{attribute 'qualified_only'}
VAR_GLOBAL
	Sc1:BOOL;
	Sc2:BOOL;
	Busc1:BOOL;
	Busc2:BOOL;
	Backup_safety_trip:BOOL;
	Main_safety_trip:BOOL;
	Lily_func_trip:BOOL;
	Lily_app_fault:BOOL;
	Backup_control_trip:BOOL;
	Control_trip:BOOL;
	Control_stop:BOOL;
	Lockout:BOOL;
	Enforced_slow:BOOL;
	Alarm:BOOL;
	All_clear:BOOL;
	Reset_button:BOOL;
	Reset_interlocks:BOOL;
	Reset:BOOL;
	Safe_for_power:BOOL;
	Bridge_present:BOOL;
END_VAR

(* stored: Version 1.1.0.1, ProductVersion 3.1.4024.0
   GVL Safety: Id {552a7057-3401-49c8-8ba8-03809ca8f408} *)
